FUNCTION_BLOCK Math
VAR_INPUT
	
END_VAR
VAR_OUTPUT
	
result		:	INT;

END_VAR
VAR
END_VAR

METHOD addition : INT
VAR_INPUT
	
input1		:	INT;
input2		:	INT;


END_VAR


result := input1 + input2;
END_METHOD

END_FUNCTION_BLOCK

(* stored: Version 1.1.0.1, ProductVersion 3.1.4024.12
   POU Math: Id {64151ea8-35af-4125-898a-d38500c1ddbb}, SpecialFunc None
   Method addition: Id {c3e6c671-af61-4a44-8435-3148136e521f} *)
